{attribute 'GeneratedUsingTerminal: EK1100-0000-0018'}
{attribute addProperty BoxType "EK1100-0000-0018"}
{attribute addProperty Id "RC40_B1_EL7041_1000EL7041_86DE63E743RC40_B2_EL7041_1000EL7041_86DE63E743RC40_C11_EL7041_1000EL7041_86DE63E743RC40_C12_EL7041_1000EL7041_86DE63E743RC40_C21_EL7041_1000EL7041_86DE63E743RC40_C22_EL7041_1000EL7041_86DE63E743RC40_2_EndTerminal_EL9010EL9010_D29C20850"}
{attribute addProperty CRC "2901440345"}
{attribute addProperty Size "258"}
{attribute addProperty Name "RC40_2 (EK1100)"}
TYPE RC40_2_EK1100_ACF07759 EXTENDS EK1100_1FC0878B :
STRUCT
	{attribute addProperty Name "RC40_B1 (EL7041-1000)"}
	{attribute addProperty PreviousPort "RC40_2 (EK1100) : B"}
	{attribute addProperty SyncUnit "C40"}
	RC40_B1_EL7041_1000 : EL7041_86DE63E7;
	{attribute addProperty Name "RC40_B2 (EL7041-1000)"}
	{attribute addProperty PreviousPort "RC40_B1 (EL7041-1000) : B"}
	{attribute addProperty SyncUnit "C40"}
	RC40_B2_EL7041_1000 : EL7041_86DE63E7;
	{attribute addProperty Name "RC40_C11 (EL7041-1000)"}
	{attribute addProperty PreviousPort "RC40_B2 (EL7041-1000) : B"}
	{attribute addProperty SyncUnit "C40"}
	RC40_C11_EL7041_1000 : EL7041_86DE63E7;
	{attribute addProperty Name "RC40_C12 (EL7041-1000)"}
	{attribute addProperty PreviousPort "RC40_C11 (EL7041-1000) : B"}
	{attribute addProperty SyncUnit "C40"}
	RC40_C12_EL7041_1000 : EL7041_86DE63E7;
	{attribute addProperty Name "RC40_C21 (EL7041-1000)"}
	{attribute addProperty PreviousPort "RC40_C12 (EL7041-1000) : B"}
	{attribute addProperty SyncUnit "C40"}
	RC40_C21_EL7041_1000 : EL7041_86DE63E7;
	{attribute addProperty Name "RC40_C22 (EL7041-1000)"}
	{attribute addProperty PreviousPort "RC40_C21 (EL7041-1000) : B"}
	{attribute addProperty SyncUnit "C40"}
	RC40_C22_EL7041_1000 : EL7041_86DE63E7;
	{attribute addProperty Name "RC40_2_EndTerminal (EL9010)"}
	{attribute addProperty PreviousPort "RC40_C22 (EL7041-1000) : B"}
	{attribute addProperty SyncUnit "default"}
	RC40_2_EndTerminal_EL9010 : EL9010_D29C2085;
END_STRUCT
END_TYPE

(* stored: Version 1.2.0.0, ProductVersion 3.1.4024.11
   DUT RC40_2_EK1100_ACF07759: Id {2bf38970-6ee2-0a94-3529-4c3e3ea1d4d9} *)
